// TIA Portal project "S7-1500 Analog Giriş ile Seviye Lambalı Su Deposu Uygulaması" (V18)

(* hardware
DEVICE "S7-1500/ET200MP station_1"  S7-1500 station
   slot 0: "Rail_0"  Rack  6ES7 590-1***0-0AA0
   slot 1: "PLC_1"  CPU 1512C-1 PN  6ES7 512-1CK01-0AB0  V2.8
      slot 3: "CPU display_1"  6ES7591-1AA00-0AA0
      slot 32768: "PROFINET interface_1"  X1
         slot 32769: "Port_1"  X1 P1
         slot 32770: "Port_2"  X1 P2
      slot 34817: "Virtual CP interface port_1"  Virtual CP interface port  Virtual CP interface port
DEVICE "HMI_1"  KTP700 Basic PN
   slot 0: "HMI_1"  KTP700 Basic PN  6AV2 123-2GB03-0AX0  14.0.1.0
   slot 1: "HMI_RT_1"  KTP700 Basic PN  6AV2 123-2GB03-0AX0  14.0.1.0
   slot 5: "HMI_1.IE_CP_1"  PROFINET Interface  14.0.1.0
      slot 1: "PROFINET Interface_1"  PROFINET Interface
         slot 1: "Port_1"  Port
*)

// ===== PLC "PLC_1"  CPU 1512C-1 PN =====

VAR_GLOBAL   // PLC tag table "Default tag table"
   "Analog Giriş" AT %IW126 : Word;
   "Analog Yardımcı" AT %MW126 : Word;
   "sayaç_1" AT %MD10 : DWord;
   "sayaç_2" AT %MW20 : Int;
   "20'den az" AT %Q0.1 : Bool;
   "20-80 arası" AT %Q0.2 : Bool;
   "80'den çok" AT %Q0.0 : Bool;
END_VAR

ORGANIZATION_BLOCK "Main"   // OB1, LAD, ProgramCycle
TITLE = "Main Program Sweep (Cycle)"
{ S7_Optimized_Access := 'TRUE' }
VERSION : 0.1
   VAR_INPUT
      Initial_Call : Bool;   // Initial call of this OB
      Remanence : Bool;   // =True, if remanent data are available
   END_VAR
BEGIN

REGION Network 1: Analog girişten alınan değeri okumak içindir.
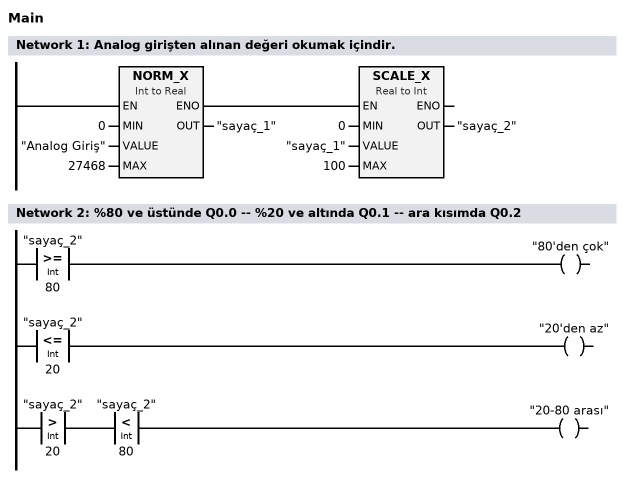
   RUNG wire#powerrail
      { S7_Templates := "[SrcType := Int, DestType := Real]" } Normalize(min := 0, value := "Analog Giriş", max := 27468, out => "sayaç_1")
      { S7_Templates := "[SrcType := Real, DestType := Int]" } Scale(min := 0, value := "sayaç_1", max := 100, out => "sayaç_2")
   END_RUNG
   // the same network as SCL:
   "sayaç_1" := NORM_X(MIN := 0, VALUE := "Analog Giriş", MAX := 27468);
   "sayaç_2" := SCALE_X(MIN := 0, VALUE := "sayaç_1", MAX := 100);
END_REGION

REGION Network 2: %80 ve üstünde Q0.0 -- %20 ve altında Q0.1 -- ara kısımda Q0.2
   RUNG wire#powerrail
      { S7_Templates := "SrcType := Int" } GE_Contact(in1 := "sayaç_2", in2 := 80)
      Coil( "80'den çok" )
   END_RUNG
   RUNG wire#powerrail
      { S7_Templates := "SrcType := Int" } LE_Contact(in1 := "sayaç_2", in2 := 20)
      Coil( "20'den az" )
   END_RUNG
   RUNG wire#powerrail
      { S7_Templates := "SrcType := Int" } GT_Contact(in1 := "sayaç_2", in2 := 20)
      { S7_Templates := "SrcType := Int" } LT_Contact(in1 := "sayaç_2", in2 := 80)
      Coil( "20-80 arası" )
   END_RUNG
   // the same network as SCL:
   "80'den çok" := "sayaç_2" >= 80;
   "20'den az" := "sayaç_2" <= 20;
   "20-80 arası" := ("sayaç_2" > 20) AND ("sayaç_2" < 80);
END_REGION
END_ORGANIZATION_BLOCK

(* ===== HMI "HMI_RT_1" =====
system functions are stored by id; their names below are inferred from use
connection "Connection_1": ETHERNET, SMART_S7_1500_OMS
connection "HMI_Connection_1": ETHERNET, SMART_S7_1500_OMS

HMI tags "Default tag table"
   "Tag_ScreenNumber" : UInt, internal
   "sayaç_2" : Int = PLC sayaç_2 AT %MW20, 100 ms
   "Doldurma Motoru_1" : Bool = PLC "20'den az" AT %Q0.1, 100 ms
   "Doldurma Motoru_2" : Bool = PLC "20-80 arası" AT %Q0.2, 100 ms
   "80den çok" : Bool = PLC "80'den çok" AT %Q0.0, 1 s

graphic list "80 den çok": 0 'Graphic_15'; 1 'Graphic_17'

graphic list "20 den az": 0 'Graphic_15'; 1 'Graphic_16'

graphic list "aralarda": 0 'Graphic_15'; 1 'Graphic_14'

Template "Template_1" 800x480
   Button "Exit" at 714,429 size 71x50; TextOff 'Exit'; PictureOff "ExitRuntime_KTP700_Basic_PN_TR"; PictureOn "ExitRuntime_KTP700_Basic_PN_TR"
      on Release: StopRuntime(0)
   Button "Language" at 614,429 size 71x50; TextOff 'Language'; PictureOff "ToggleLanguage_KTP700_Basic_PN_TR"; PictureOn "ToggleLanguage_KTP700_Basic_PN_TR"
      on Release: function_fb9197e8(-1)
   Button "Log on" at 514,429 size 71x50; TextOff 'Log on'; PictureOff "Login_KTP700_Basic_PN_TR"; PictureOn "Login_KTP700_Basic_PN_TR"
      on Release: function_a2a04561()
   Button "Alarms" at 114,429 size 71x50; TextOff 'Alarms'; PictureOff "AlarmDisplay_KTP700_Basic_PN_TR"; PictureOn "AlarmDisplay_KTP700_Basic_PN_TR"
      on Release: function_ef3f5d25("Alarm window_Unacknowledged", -1)
   Button "Start screen" at 14,429 size 71x50; TextOff 'Start screen'; PictureOff "NavigateHome_KTP700_Basic_PN_TR"; PictureOn "NavigateHome_KTP700_Basic_PN_TR"
      on Release: ActivateScreen("Root screen", 0)
   SymbolicIOField "Symbolic_IO_Field_Screen" at 93,9 size 600x33; TextOff '0'; TextOn '1'; TextList "TextList_ScreenNames"
      ProcessValue <- "Tag_ScreenNumber"
      on Change: ActivateScreenByNumber("Tag_ScreenNumber", 0)
   DateTimeField "HmiScreenItemData" at 695,25 size 105x25
   DateTimeField "HmiScreenItemData_1" at 695,0 size 105x25
   GraphicView "Logo" at 0,0 size 91x51; Picture "Logo of HMI_1"

screen "Root screen" 800x480, template "Template_1"
   on GenerateScreen: SetTag("Tag_ScreenNumber", 1)
   Bar "Bar_1" at 57,159 size 118x240; MinimumValue 0; MaximumValue 100
      ProcessValue <- "sayaç_2"
   IOField "I/O field_1" at 57,73 size 117x78; FormatPattern s99999
      ProcessValue <- "sayaç_2"
   GraphicIOField "Graphic I/O field_1" at 220,159 size 96x59; PictureList "80 den çok"
      ProcessValue <- "80den çok"
   GraphicIOField "Graphic I/O field_2" at 220,338 size 96x56; PictureList "20 den az"
      ProcessValue <- "Doldurma Motoru_1"
   GraphicIOField "Graphic I/O field_3" at 219,252 size 96x59; PictureList "aralarda"
      ProcessValue <- "Doldurma Motoru_2"
*)